{attribute 'GeneratedUsingTerminal: AT2025-0250-0023'}
{attribute addProperty BoxType "AT2025-0250-0023"}
{attribute addProperty Id "A_0076_AT2001_5250_0017_AT2001_5250AT2001_01D6DEDF80"}
{attribute addProperty CRC "466651952"}
{attribute addProperty Size "80"}
TYPE A_0064_AT2025_0250_0023_AT2025_0250_1BD08B30 EXTENDS AT2025_86175B41 :
STRUCT
	{attribute addProperty Name "A_0076_AT2001_5250_0017_AT2001_5250"}
	{attribute addProperty PreviousPort "A_0064(AT2025-0250-0023) (AT2025-0250) : B"}
	A_0076_AT2001_5250_0017_AT2001_5250 : AT2001_01D6DEDF;
END_STRUCT
END_TYPE

(* stored: Version 1.2.0.0, ProductVersion 3.1.4024.9
   DUT A_0064_AT2025_0250_0023_AT2025_0250_1BD08B30: Id {5881144d-2029-4587-8486-a89e04b07833} *)
